{attribute 'qualified_only'}
TYPE E_BiaxialState :
(
	Idle,
	Running,
	Aborting,
	Completing
);
END_TYPE

(* stored: Version 1.1.0.1, ProductVersion 3.1.4024.15
   DUT E_BiaxialState: Id {a3af55a7-38d1-4b18-a50e-81382a2277d1} *)
